FUNCTION_BLOCK FB_LightDimmIndirectNC
VAR_INPUT
	bInputs				:	ARRAY[0..nSize] OF BOOL;	//Input Schalter oder Taster
	bInputSec			:	BOOL := FALSE;				//Input für Security Schaltung
	bInputSecTest		:	BOOL := FALSE;				//Testeingang für den Sec Modus
	bAllFlanks			:	BOOL := FALSE;				//Alle Flanken verwenden?
	tLongPress			:	TIME := T#1000MS;			//Long Press Zeit für AUS!
	tBlockTime			:	TIME := T#2000MS;			//Zeit nach Ausschalten bis wiedereinschalten
	iNumPress4Dimm		:	UINT := 4;					//Reduktion der Helligkeit je Tastendruck
END_VAR
VAR_IN_OUT
	bInputHA		:	BOOL;						//Input (HA)
	iDimmValue		:	WORD;						//DimmValue Input
END_VAR
VAR_OUTPUT
	iOut			:	INT;
	bOut			:	BOOL;
END_VAR
VAR CONSTANT
	nSize 			:	UINT := 5; 					//Maximale Anzahl Eingänge
END_VAR
VAR
	fbRtrig			:	ARRAY[0..nSize] OF R_TRIG;
	fbFtrig			:	ARRAY[0..nSize] OF F_TRIG;
	tonLongPress	:	ARRAY[0..nSize] OF TON;
	tonBlock		:	TON;
	
	Idx				:	UINT;
	
	bSecRising		:	BOOL := TRUE;
	bBlock			:	BOOL := FALSE;

END_VAR
VAR_TEMP
	iCountDimm		:	UINT;
	iCalcReduction	:	INT;
	
	bTrigger		:	BOOL := FALSE;
	bAllOFF			:	BOOL := FALSE;
END_VAR


tonBlock(IN := bBlock, PT := tBlockTime);

IF tonBlock.Q THEN
	bBlock	:= FALSE;
END_IF

IF (bInputSec OR bInputSecTest) AND NOT bBlock THEN	//Party bei Security Falls
	
	bInputHA	:= TRUE;
	bOut		:= FALSE;		// !!! NC
	
	IF bSecRising THEN
		
		iDimmValue := iDimmValue + 5;

		IF iDimmValue = 255 THEN
			bSecRising := FALSE;
		END_IF	
	
	ELSE
	
		iDimmValue := iDimmValue - 5;

		IF iDimmValue <= 0 THEN
			bSecRising := TRUE;
		END_IF	
	
	END_IF

	
ELSE	//Normale Funktion

	//Init alle Flankentrigger und Frage diese ab
	FOR Idx := 0 TO nSize DO
	
		//Alle R_Trig
		fbRtrig[Idx](CLK:= bInputs[Idx], Q=> );
		tonLongPress[Idx](IN := bInputs[Idx], PT := tLongPress);
		
		bTrigger := bTrigger OR fbRtrig[Idx].Q;
		bAllOFF	:= bAllOFF OR tonLongPress[Idx].Q;
	
		IF bAllFlanks THEN //Wenn alle Flanken
			fbFtrig[Idx](CLK:= bInputs[Idx], Q=> );
			bTrigger := bTrigger OR fbFtrig[Idx].Q;
		END_IF
	
	END_FOR

	IF (iDimmValue > 0 OR bInputHA) AND iOut = 0 AND NOT bBlock THEN		//Wenn über HA Eingeschaltet
		bInputHA	:= TRUE;
		bOut		:= FALSE;		// !!! NC
		
		IF iDimmValue = 0 THEN
			iDimmValue	:= 255;
		END_IF
	END_IF
	
	IF bTrigger AND NOT bBlock THEN
		
		IF iOut = 0 THEN					//Erstes Einschalten über Schalter
			bInputHA	:= TRUE;
			bOut		:= FALSE;			// !!! NC
			iDimmValue	:= 255;
		
		ELSE
			
			FOR iCountDimm := 0 TO iNumPress4Dimm DO
			
			iCalcReduction := (256 - (iCountDimm * (256 / iNumPress4Dimm)));
		
			IF iDimmValue > iCalcReduction THEN
				iDimmValue := iCalcReduction;
				EXIT;
			END_IF
		
			END_FOR
		
		END_IF
		
	END_IF

END_IF

IF bAllOFF OR bInputHA = FALSE OR iDimmValue <= 0 THEN		//Alles Ausschalten
	bInputHA	:= FALSE;
	bOut		:= TRUE;			// !!! NC
	iDimmValue	:= 0;
	bBlock		:= TRUE;
END_IF

iOut := F_LightDimmingConvertForHA(iDimmValue);

END_FUNCTION_BLOCK

(* stored: Version 1.1.0.1, ProductVersion 3.1.4024.4
   POU FB_LightDimmIndirectNC: Id {27ce8e36-3e5a-49e5-985e-127cbdb4bf8b}, SpecialFunc None *)
